TYPE VelocityCtrl_Input_typ :
	STRUCT
		Command 	: VelocityCtrl_CMD_typ ;
		Parameter	: VelocityCtrl_Param_typ ;
	END_STRUCT
END_TYPE

(* stored: Version 1.1.0.1, ProductVersion 3.1.4024.3
   DUT VelocityCtrl_Input_typ: Id {0e3d8da6-b606-4cc0-a499-d5928b62dbe9} *)
